# EPICS autosave request: iocBoot/iocLTC2983/autosave/pv-spi01-a.req
$(SNAME):CH8:if
